// TwinCAT 3 PLC project PubSubSampleProject_Publisher
// ProgramVersion: 3.1.4026.1+c9eadab3edd020c56c333d811d5b3c408c2550c8
// libraries:
//   Tc2_Standard, * (Beckhoff Automation GmbH)
//   Tc2_System, * (Beckhoff Automation GmbH)
// project tree:
//   DUTs/ ST_MyStructure.TcDUT (not stored)
//   GVLs/ GVL_PublisherVars_1.TcGVL (not stored), GVL_PublisherVars_2.TcGVL (not stored)
//   / PlcTask.TcTTO
//   POUs/ MAIN.TcPOU
// real-time tasks:
//   TASK PlcTask: cycle T#10ms, priority 20, ADS port 350
//   TASK PlcTask1: cycle T#10ms, priority 21, ADS port 351
// I/O:
//   DEVICE Device 1 (OPC UA RT), AmsNetId 172.16.71.15.2.1
// variable links:
//   PubSubSampleProject_Publisher/PubSubSampleProject_Publisher Instance <-> Device 1 (OPC UA RT)/Publisher1/DsPubVars1
//     PlcTask Outputs/GVL_PublisherVars_1.nCounter <-> Outputs/GVL_PublisherVars_1_nCounter
//     PlcTask Outputs/GVL_PublisherVars_1.sString <-> Outputs/GVL_PublisherVars_1_sString
//     PlcTask Outputs/GVL_PublisherVars_1.stMyStruct <-> Outputs/GVL_PublisherVars_1_stMyStruct
//   PubSubSampleProject_Subscriber/PubSubSampleProject_Subscriber Instance <-> Device 1 (OPC UA RT)/Subscriber1/DsPubVars1
//     PlcTask Inputs/GVL_SubscriberVars_1.nCounter <-> Inputs/GVL_PublisherVars_1_nCounter
//     PlcTask Inputs/GVL_SubscriberVars_1.sString <-> Inputs/GVL_PublisherVars_1_sString
//     PlcTask Inputs/GVL_SubscriberVars_1.stMyStruct <-> Inputs/GVL_PublisherVars_1_stMyStruct
//   PubSubSampleProject_Subscriber/PubSubSampleProject_Subscriber Instance <-> Device 1 (OPC UA RT)/Subscriber2/DsPub1
//     PlcTask Inputs/GVL_SubscriberVars_2.nCounter <-> Inputs/GVL_PublisherVars_2_nCounter
//     PlcTask Inputs/GVL_SubscriberVars_2.sString <-> Inputs/GVL_PublisherVars_2_sString
//     PlcTask Inputs/GVL_SubscriberVars_2.stMyStruct <-> Inputs/GVL_PublisherVars_2_stMyStruct

CONFIGURATION PubSubSampleProject_Publisher
    RESOURCE PLC ON TwinCAT3
        TASK PlcTask(INTERVAL := T#10ms, PRIORITY := 20);
        PROGRAM MAIN WITH PlcTask : MAIN;
    END_RESOURCE
END_CONFIGURATION

// ---- POUs/MAIN.TcPOU
(* This sample demonstrates how to configure TF6105 OPC UA Pub/Sub with a publisher and a subscriber. This PLC Project contains the publisher.
   The publisher comes in two flavors: one publisher that contains a data set WITH process image variables and one publisher that contains a 
   data set WITHOUT process image variables. In this case the variables are mapped internally to the corresponding ADS symbol names. This can
   be achieved by using the TwinCAT Target Browser to drag&drop variables onto the data set fields of the data set. 

   The publishers on the OPC UA RT device have been set up manually whereas the corresponding subscribers have been set up by using the 
   OPC UA Binary exchange file.

   Please consult our documentation on the Beckhoff Information System for more information. *)
PROGRAM MAIN
VAR
END_VAR

(* Update publisher variables 1 with random values *)
GVL_PublisherVars_1.sString := CONCAT('Hello World ', TO_STRING(GVL_PublisherVars_1.nCounter));
GVL_PublisherVars_1.stMyStruct.a := GVL_PublisherVars_1.stMyStruct.a + 1;
GVL_PublisherVars_1.stMyStruct.b := GVL_PublisherVars_1.stMyStruct.b + 1;
GVL_PublisherVars_1.stMyStruct.c := GVL_PublisherVars_1.stMyStruct.c + 0.1;
GVL_PublisherVars_1.stMyStruct.d := CONCAT('Hello World ', TO_STRING(GVL_PublisherVars_1.nCounter));
GVL_PublisherVars_1.nCounter := GVL_PublisherVars_1.nCounter + 1;

(* Update publisher variables 2 with random values *)
GVL_PublisherVars_2.sString := CONCAT('Hello World ', TO_STRING(GVL_PublisherVars_2.nCounter));
GVL_PublisherVars_2.stMyStruct.a := GVL_PublisherVars_2.stMyStruct.a + 1;
GVL_PublisherVars_2.stMyStruct.b := GVL_PublisherVars_2.stMyStruct.b + 1;
GVL_PublisherVars_2.stMyStruct.c := GVL_PublisherVars_2.stMyStruct.c + 0.1;
GVL_PublisherVars_2.stMyStruct.d := CONCAT('Hello World ', TO_STRING(GVL_PublisherVars_2.nCounter));
GVL_PublisherVars_2.nCounter := GVL_PublisherVars_2.nCounter + 1;

END_PROGRAM
